PROGRAM POU
VAR
	test:BOOL;
END_VAR

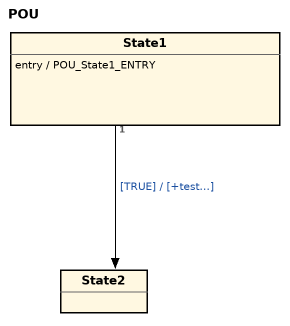
STATECHART POU  // abortable
    STATE State1
        entry / POU_State1_ENTRY
    STATE State2
    State1 -> State2 [TRUE] / [+test...] // priority 1
END_STATECHART

ACTION POU_State1_ENTRY:

END_ACTION

END_PROGRAM

(* stored: Version 1.1.0.1, ProductVersion 3.1.4024.3
   POU POU: Id {287c4922-88fc-464d-8a45-4246dd669713}, SpecialFunc None
   Action POU_State1_ENTRY: Id {db416b4a-c7cb-4ab6-995e-a7445f93f614} *)
